FUNCTION_BLOCK FB_ModeVisualization
VAR_INPUT
END_VAR
VAR_OUTPUT
END_VAR
VAR
END_VAR

METHOD Auto
VAR_INPUT
	bEnable : BOOL;
END_VAR
IF bEnable THEN
	G_VB.eMode := E_Mode.Auto;
END_IF
END_METHOD

METHOD Manual
VAR_INPUT
	bEnable : BOOL;
END_VAR
IF bEnable THEN
	G_VB.eMode := E_Mode.Manual;
END_IF
END_METHOD

METHOD Off
VAR_INPUT
	bEnable : BOOL;
END_VAR
IF bEnable THEN
	G_VB.eMode := E_Mode.OFF;
END_IF
END_METHOD

END_FUNCTION_BLOCK

(* stored: Version 1.1.0.1, ProductVersion 3.1.4024.12
   POU FB_ModeVisualization: Id {6974c941-443e-4297-a4bf-0fa9ebcac1c2}, SpecialFunc None
   Method Auto: Id {5c1f72fd-a66d-45be-ade5-39c0e8007b91}
   Method Manual: Id {0bda4b34-43ce-47cd-ac2f-d3c89dac0863}
   Method Off: Id {7a42fcde-312e-486f-9962-b7fdafd495cd} *)
